(* IEC 61131-3 sources: CPSForge/configs/openplc, 3 files *)

(* ---- level_control.st ---- *)
(* =============================================================================
   CPSForge — Level Control for OpenPLC
   =============================================================================
   Structured Text for OpenPLC Runtime v4 (matiec-compatible).

   All located variables use %QW (holding registers) or %QX (coils) so
   both the PLC and the Modbus simulator can read/write them.
   No %IX or %IW (those are read-only via Modbus).

   Analog values are scaled x100: physical = raw_int * 0.01
     (e.g., 500 = 5.00 V, 1000 = 10.00 V)

   Modbus register mapping:
     %QW0  : FillValve      (INT x100, 0-1000)
     %QW1  : DischargeValve (INT x100, 0-1000)
     %QW2  : SPDisplay      (INT x100, mirror of setpoint)
     %QW3  : PVDisplay      (INT x100, mirror of level)
     %QW10 : LevelMeter     (INT x100, simulator writes)
     %QW11 : FlowMeter      (INT x100, simulator writes)
     %QW12 : SetpointIn     (INT x100, default 500, attackable)
     %QX0.0 : Running       (auto-True when Enable)
     %QX0.1 : Enable        (kill switch, default TRUE)
   ============================================================================= *)

PROGRAM level_control
  VAR
    (* Sensor inputs — written by simulator via Modbus holding registers *)
    LevelMeter_raw  AT %QW10 : INT := 0;
    FlowMeter_raw   AT %QW11 : INT := 0;
    SetpointIn_raw  AT %QW12 : INT := 500;

    (* Actuator outputs — computed by this program *)
    FillValve_raw       AT %QW0 : INT := 0;
    DischargeValve_raw  AT %QW1 : INT := 0;
    SPDisplay_raw       AT %QW2 : INT := 0;
    PVDisplay_raw       AT %QW3 : INT := 0;

    (* Digital state *)
    Running     AT %QX0.0 : BOOL := FALSE;
    Enable      AT %QX0.1 : BOOL := TRUE;
  END_VAR
  VAR
    (* Internal temps for integer math *)
    err      : INT;
    out_val  : INT;
  END_VAR

  (* Safety gate: if Enable is FALSE, shut everything down *)
  IF NOT Enable THEN
    FillValve_raw := 0;
    DischargeValve_raw := 1000;
    Running := FALSE;
    SPDisplay_raw := 0;
    PVDisplay_raw := LevelMeter_raw;
    RETURN;
  END_IF;

  (* Auto-run when enabled — no physical button logic needed *)
  Running := TRUE;

  (* Update displays *)
  SPDisplay_raw := SetpointIn_raw;
  PVDisplay_raw := LevelMeter_raw;

  (* Proportional control — all in INT x100 space *)
  err := SetpointIn_raw - LevelMeter_raw;

  IF err > 0 THEN
    out_val := err;
    IF out_val > 1000 THEN out_val := 1000; END_IF;
    FillValve_raw := out_val;
    DischargeValve_raw := 0;
  ELSE
    FillValve_raw := 0;
    out_val := -err;
    IF out_val > 1000 THEN out_val := 1000; END_IF;
    DischargeValve_raw := out_val;
  END_IF;

END_PROGRAM

CONFIGURATION Config0
  RESOURCE Res0 ON PLC
    TASK Main(INTERVAL := T#50ms, PRIORITY := 0);
    PROGRAM Inst0 WITH Main : level_control;
  END_RESOURCE
END_CONFIGURATION

(* ---- sorting_height.st ---- *)
(* =============================================================================
   CPSForge — Sorting by Height Basic (OpenPLC Structured Text)
   =============================================================================
   IEC 61131-3 Structured Text for OpenPLC Runtime v4 (matiec-compatible).

   2-way height sorter:
     Short item (low sensor only) -> Transfer LEFT
     Tall  item (high sensor)     -> Transfer RIGHT

   State machine:
     0=Feed, 1=Load, 2=Transfer, 3=Clear, 4=Finish

   ALL located variables use %QW (holding registers) or %QX (coils) so
   both PLC and Modbus simulator can read/write them.
   No %IX or %IW (read-only via Modbus).

   Modbus mapping:
     Actuator outputs (Holding Registers):
       HR0-%QW0   ConveyorEntry   HR4-%QW4   TransfRight
       HR1-%QW1   LoadAct         HR5-%QW5   ConveyorLeft
       HR2-%QW2   UnloadAct       HR6-%QW6   ConveyorRight
       HR3-%QW3   TransfLeft

     Counters/state (Holding Registers):
       HR10-%QW10  CounterOut      HR11-%QW11  iState

     Mode (Coils):
       COIL0-%QX0.0  Enable

     Sensor inputs from simulator (Coils):
       COIL8-%QX1.0   HighSensor      COIL12-%QX1.4  AtLeftEntry
       COIL9-%QX1.1   LowSensor       COIL13-%QX1.5  AtLeftExit
       COIL10-%QX1.2  PalletSensor    COIL14-%QX1.6  AtRightEntry
       COIL11-%QX1.3  Loaded          COIL15-%QX1.7  AtRightExit
   ============================================================================= *)

PROGRAM SortingHeight
  VAR
    (* Actuator outputs — Holding Registers *)
    ConveyorEntry   AT %QW0   : INT := 0;
    LoadAct         AT %QW1   : INT := 0;
    UnloadAct       AT %QW2   : INT := 0;
    TransfLeft      AT %QW3   : INT := 0;
    TransfRight     AT %QW4   : INT := 0;
    ConveyorLeft    AT %QW5   : INT := 0;
    ConveyorRight   AT %QW6   : INT := 0;

    (* Counters + state — Holding Registers *)
    CounterOut      AT %QW10  : INT := 0;
    iState          AT %QW11  : INT := 0;

    (* Mode — Coils *)
    Enable          AT %QX0.0 : BOOL := TRUE;

    (* Sensor inputs from simulator — Coils (writable via Modbus) *)
    HighSensor      AT %QX1.0 : BOOL := FALSE;
    LowSensor       AT %QX1.1 : BOOL := FALSE;
    PalletSensor    AT %QX1.2 : BOOL := FALSE;
    Loaded          AT %QX1.3 : BOOL := FALSE;
    AtLeftEntry     AT %QX1.4 : BOOL := FALSE;
    AtLeftExit      AT %QX1.5 : BOOL := FALSE;
    AtRightEntry    AT %QX1.6 : BOOL := FALSE;
    AtRightExit     AT %QX1.7 : BOOL := FALSE;
  END_VAR
  VAR
    (* Internal — non-located *)
    IsTall          : BOOL := FALSE;
    DwellTimer      : INT  := 0;
    ItemCount       : INT  := 0;
  END_VAR

  (* ── Safety gate ── *)
  IF NOT Enable THEN
    ConveyorEntry := 0; LoadAct := 0; UnloadAct := 0;
    TransfLeft := 0; TransfRight := 0;
    ConveyorLeft := 0; ConveyorRight := 0;
    RETURN;
  END_IF;

  (* Exit conveyors always ON *)
  ConveyorLeft  := 1;
  ConveyorRight := 1;

  (* ── State machine ── *)
  CASE iState OF
    0: (* FEED: entry conveyor on, detect height *)
      ConveyorEntry := 1;
      LoadAct := 0; UnloadAct := 0;
      TransfLeft := 0; TransfRight := 0;

      IF HighSensor THEN IsTall := TRUE;
      ELSIF LowSensor THEN IsTall := FALSE;
      END_IF;

      IF PalletSensor THEN
        DwellTimer := 0;
        iState := 1;
      END_IF;

    1: (* LOAD: run entry conveyor until loaded *)
      IF Loaded THEN ConveyorEntry := 0;
      ELSE ConveyorEntry := 1;
      END_IF;
      LoadAct := 1;
      UnloadAct := 0;
      TransfLeft := 0; TransfRight := 0;

      IF HighSensor THEN IsTall := TRUE;
      ELSIF LowSensor THEN IsTall := FALSE;
      END_IF;

      DwellTimer := DwellTimer + 1;

      IF Loaded THEN
        DwellTimer := 0;
        iState := 2;
      ELSIF DwellTimer > 5000 THEN
        ConveyorEntry := 0;
        DwellTimer := 0;
        iState := 2;
      END_IF;

    2: (* TRANSFER: short->LEFT, tall->RIGHT *)
      ConveyorEntry := 0;
      LoadAct := 1;  (* Keep chains raised *)

      IF IsTall THEN
        TransfRight := 1; TransfLeft := 0;
      ELSE
        TransfLeft := 1; TransfRight := 0;
      END_IF;

      DwellTimer := DwellTimer + 1;
      IF DwellTimer > 3000 THEN
        DwellTimer := 0;
        iState := 3;
      END_IF;

    3: (* CLEAR: wait for item to leave *)
      ConveyorEntry := 0;
      LoadAct := 0;
      UnloadAct := 1;
      TransfLeft := 0; TransfRight := 0;

      DwellTimer := DwellTimer + 1;
      IF DwellTimer > 2000 THEN
        DwellTimer := 0;
        iState := 4;
      END_IF;

    4: (* FINISH: increment counter, return to feed *)
      UnloadAct := 0;
      ItemCount := ItemCount + 1;
      CounterOut := ItemCount;
      iState := 0;

  ELSE
    iState := 0;
  END_CASE;

END_PROGRAM

CONFIGURATION Config0
  RESOURCE Res0 ON PLC
    TASK Main(INTERVAL := T#50ms, PRIORITY := 0);
    PROGRAM Inst0 WITH Main : SortingHeight;
  END_RESOURCE
END_CONFIGURATION

(* ---- sorting_weight.st ---- *)
(* =============================================================================
   CPSForge — Sorting by Weight (OpenPLC Structured Text)
   =============================================================================
   IEC 61131-3 Structured Text for OpenPLC Runtime v4 (matiec-compatible).

   3-way weight sorter: weigh each box on a scale, then route:
     weight < LightThresh (200 = 2.0 kg) -> LEFT
     weight >= HeavyThresh (500 = 5.0 kg) -> RIGHT
     otherwise -> FORWARD

   ALL located variables use %QW (holding registers) or %QX (coils) so
   both PLC and Modbus simulator can read/write them.
   No %IX or %IW (read-only via Modbus).

   Modbus mapping:
     Actuator outputs (Holding Registers):
       HR0-%QW0  EntryConveyor     HR4-%QW4  SendRight
       HR1-%QW1  LoadScale         HR5-%QW5  RightConveyor
       HR2-%QW2  SendLeft          HR6-%QW6  SendForward
       HR3-%QW3  LeftConveyor      HR7-%QW7  FrontConveyor

     Thresholds/state (Holding Registers, INT x100):
       HR10-%QW10  LightThresh     HR12-%QW12  MeasuredWeight
       HR11-%QW11  HeavyThresh     HR13-%QW13  Weight_raw (sim writes)

     Counters (Holding Registers):
       HR20-%QW20  LeftCount       HR22-%QW22  RightCount
       HR21-%QW21  ForwardCount    HR23-%QW23  iState

     Mode/state (Coils):
       COIL0-%QX0.0  Enable

     Sensor inputs from simulator (Coils):
       COIL8-%QX1.0   AtScaleEntry    COIL13-%QX1.5  AtForwardEntry
       COIL9-%QX1.1   AtScale         COIL14-%QX1.6  AtExitFront
       COIL10-%QX1.2  AtScaleExit     COIL15-%QX1.7  AtRightEntry
       COIL11-%QX1.3  AtLeftEntry     COIL16-%QX2.0  AtExitRight
       COIL12-%QX1.4  AtExitLeft
   ============================================================================= *)

PROGRAM SortingWeight
  VAR
    (* Actuator outputs — Holding Registers *)
    EntryConveyor   AT %QW0   : INT := 0;
    LoadScale       AT %QW1   : INT := 0;
    SendLeft        AT %QW2   : INT := 0;
    LeftConveyor    AT %QW3   : INT := 0;
    SendRight       AT %QW4   : INT := 0;
    RightConveyor   AT %QW5   : INT := 0;
    SendForward     AT %QW6   : INT := 0;
    FrontConveyor   AT %QW7   : INT := 0;

    (* Thresholds — Holding Registers (INT x100) *)
    LightThresh     AT %QW10  : INT := 200;
    HeavyThresh     AT %QW11  : INT := 500;
    MeasuredWeight  AT %QW12  : INT := 0;

    (* Weight sensor — simulator writes here via Modbus HR13 *)
    Weight_raw      AT %QW13  : INT := 0;

    (* Counters + state — Holding Registers *)
    LeftCount       AT %QW20  : INT := 0;
    ForwardCount    AT %QW21  : INT := 0;
    RightCount      AT %QW22  : INT := 0;
    iState          AT %QW23  : INT := 0;

    (* Mode — Coils *)
    Enable          AT %QX0.0 : BOOL := TRUE;

    (* Sensor inputs from simulator — Coils (writable via Modbus) *)
    AtScaleEntry    AT %QX1.0 : BOOL := FALSE;
    AtScale         AT %QX1.1 : BOOL := FALSE;
    AtScaleExit     AT %QX1.2 : BOOL := FALSE;
    AtLeftEntry     AT %QX1.3 : BOOL := FALSE;
    AtExitLeft      AT %QX1.4 : BOOL := FALSE;
    AtForwardEntry  AT %QX1.5 : BOOL := FALSE;
    AtExitFront     AT %QX1.6 : BOOL := FALSE;
    AtRightEntry    AT %QX1.7 : BOOL := FALSE;
    AtExitRight     AT %QX2.0 : BOOL := FALSE;
  END_VAR

  (* Exit conveyors always run *)
  LeftConveyor  := 1;
  FrontConveyor := 1;
  RightConveyor := 1;

  (* Default thresholds if not set *)
  IF LightThresh < 10 THEN LightThresh := 200; END_IF;
  IF HeavyThresh < 10 THEN HeavyThresh := 500; END_IF;

  IF NOT Enable THEN
    EntryConveyor := 0;
    LoadScale     := 0;
    SendLeft      := 0;
    SendRight     := 0;
    SendForward   := 0;
    iState        := 0;
  ELSE
    CASE iState OF
      0: (* Idle — feed box onto scale *)
        EntryConveyor := 1;
        LoadScale     := 1;
        SendLeft      := 0;
        SendRight     := 0;
        SendForward   := 0;
        IF AtScale THEN
          EntryConveyor := 0;
          LoadScale     := 0;
          MeasuredWeight := Weight_raw;
          iState := 1;
        END_IF;

      1: (* Weighed — decide direction *)
        EntryConveyor := 0;
        LoadScale     := 0;
        IF MeasuredWeight < LightThresh THEN
          SendLeft := 1;
          iState := 2;
        ELSIF MeasuredWeight >= HeavyThresh THEN
          SendRight := 1;
          iState := 4;
        ELSE
          SendForward := 1;
          iState := 6;
        END_IF;

      2: (* Sending left *)
        SendLeft  := 1;
        LoadScale := 1;
        IF NOT AtScale AND NOT AtScaleExit THEN
          SendLeft    := 0;
          LoadScale   := 0;
          LeftCount   := LeftCount + 1;
          iState      := 0;
        END_IF;

      4: (* Sending right *)
        SendRight := 1;
        LoadScale := 1;
        IF NOT AtScale AND NOT AtScaleExit THEN
          SendRight   := 0;
          LoadScale   := 0;
          RightCount  := RightCount + 1;
          iState      := 0;
        END_IF;

      6: (* Sending forward *)
        SendForward := 1;
        LoadScale   := 1;
        IF NOT AtScale AND NOT AtScaleExit THEN
          SendForward  := 0;
          LoadScale    := 0;
          ForwardCount := ForwardCount + 1;
          iState       := 0;
        END_IF;

    ELSE
      iState := 0;
    END_CASE;
  END_IF;

END_PROGRAM

CONFIGURATION Config0
  RESOURCE Res0 ON PLC
    TASK Main(INTERVAL := T#50ms, PRIORITY := 0);
    PROGRAM Inst0 WITH Main : SortingWeight;
  END_RESOURCE
END_CONFIGURATION
